(* CODESYS project mobject-graph-plc-pack.library
   Company: mobject
   DefaultNamespace: mobject-graph-plc-pack
   Version: 0.17.0
   Placeholder: mobject-graph-plc-pack
   Author: mobject dev team
   Title: mobject-graph-plc-pack

Project tree, tasks and I/O mapping:
  libraries: mobject-core, 0.7.0 (mobject); mobject-graph, 0.16.0 (mobject); Tc2_Standard, * (Beckhoff Automation GmbH); Tc2_System, * (Beckhoff Automation GmbH); Tc2_Utilities, * (Beckhoff Automation GmbH); Tc3_Module, * (Beckhoff Automation GmbH)
  Datatypes/
    Alias/
      function block _FLOAT [ST]: SetBaseDatatypeReference, Address, ClearReference, Size, FB_init, Clone, Identifier, MakeReferenceTo, TryMakeReferenceTo, Value
      function block _HRESULT [ST]: SetBaseDatatypeReference, Address, ClearReference, Size, FB_init, Clone, Identifier, MakeReferenceTo, TryMakeReferenceTo, Value
    Arrays/
      function block _Array0To7OfByte [ST]: FB_init, OnSerializeArrayValues, SetElementReference, TryDeserializeArrayValues, Address, BaseDatatype, ClearReference, Size, TryGetElementAsDatatypeByIndex, TryGetLowerBound, TryGetUpperBound, Clone, MakeReferenceTo, TryMakeReferenceTo, Value
    Enums/
      function block _E_TcEventClass [ST]: SetBaseDatatypeReference, Address, ClearReference, Size, FB_init, AddLocalEnumeration, IsEnumeratorValueEqual, Clone, Identifier, MakeReferenceTo, TryMakeReferenceTo, Value
    Structs/
      function block _GUID [ST]: Address, ClearReference, Size, FB_init, SetMemberReference, Clone, Identifier, IsValidGuidString, MakeReferenceTo, TryDeserializeFrom, TryMakeReferenceTo, Value, Data1, Data2, Data3, Data4, ToString, TryFromString
      function block _TIMESTRUCT [ST]: Address, ClearReference, Size, FB_init, SetMemberReference, Clone, Identifier, MakeReferenceTo, TryMakeReferenceTo, Value, wDay, wDayOfWeek, wHour, wMilliseconds, wMinute, wMonth, wSecond, wYear
    function block PlcDatatypePack [ST]: RegisterWithDatatypes
  Nodes/
    Converter/
      BOOL_TO_/
      BYTE_TO_/
      DATE_TO_/
      DINT_TO_/
        function block Node_DINT_TO_LREAL [ST]: FB_init, Clone, OnExecute
        function block Node_DINT_TO_REAL [ST]: FB_init, Clone, OnExecute
      DT_TO_/
      DWORD_TO_/
      INT_TO_/
      LINT_TO_/
      LREAL_TO_/
        function block Node_LREAL_TO_DINT [ST]: FB_init, Clone, OnExecute
        function block Node_LREAL_TO_UDINT [ST]: FB_init, Clone, OnExecute
      LWORD_TO_/
      REAL_TO_/
        function block Node_REAL_TO_DINT [ST]: FB_init, Clone, OnExecute
        function block Node_REAL_TO_UDINT [ST]: FB_init, Clone, OnExecute
      SINT_TO_/
      STRING_TO_/
      TIME_TO_/
      TOD_TO_/
      UDINT_TO_/
        function block Node_UDINT_TO_LREAL [ST]: FB_init, Clone, OnExecute
        function block Node_UDINT_TO_REAL [ST]: FB_init, Clone, OnExecute
      UINT_TO_/
      ULINT_TO_/
      USINT_TO_/
      WORD_TO_/
    Hardware/
      Digital/
        function block Node_DigitalInput [ST]: FB_init, OnExecute
        function block Node_DigitalOutput [ST]: FB_init, OnExecute
    Logic/
      function block Node_AND [ST]: FB_init, Clone, OnExecute
      function block Node_NAND [ST]: FB_init, Clone, OnExecute
      function block Node_NOR [ST]: FB_init, Clone, OnExecute
      function block Node_NOT [ST]: FB_init, Clone, OnExecute
      function block Node_OR [ST]: FB_init, Clone, OnExecute
      function block Node_XNOR [ST]: FB_init, Clone, OnExecute
      function block Node_XOR [ST]: FB_init, Clone, OnExecute
    TwinCAT/
      function block Node_TwinCATStatus [ST]: FB_init, Clone, OnExecute
    function block PlcNodePack [ST]: RegisterWithNodeFactory
  function block PlcPack [ST]: Register
*)

// Datatypes/Alias/_FLOAT
{attribute 'linkalways'} 
{attribute 'no_explicit_call' := 'This FB is a CLASS and must be accessed using methods or properties'}
{attribute 'enable_dynamic_creation'}
FUNCTION_BLOCK _FLOAT EXTENDS AliasDatatypeBase
VAR
	localData : FLOAT;
	activeData : REFERENCE TO FLOAT REF= localData;
	aliasBaseDatatype : _LREAL(localData);
END_VAR

METHOD PROTECTED SetBaseDatatypeReference
VAR_INPUT
END_VAR
aliasBaseDatatype.MakeReferenceTo(activeData);
END_METHOD

PROPERTY PUBLIC Address : PVOID
GET
Address := ADR(activeData);
END_GET
END_PROPERTY

METHOD PUBLIC ClearReference
VAR_INPUT
END_VAR
activeData REF= localData;
SetBaseDatatypeReference();
END_METHOD

PROPERTY PUBLIC Size : UDINT
GET
Size := SIZEOF(activeData);
END_GET
END_PROPERTY

METHOD FB_init : BOOL
VAR_INPUT
	bInitRetains : BOOL; // if TRUE, the retain variables are initialized (warm start / cold start)
	bInCopyCode : BOOL;  // if TRUE, the instance afterwards gets moved into the copy code (online change)
	InitialValue : FLOAT;
END_VAR
localData := InitialValue;
SetBaseDatatypeReference();
AddBaseDatatype(aliasBaseDatatype);
END_METHOD

METHOD PUBLIC Clone : I_Datatype
VAR
    pClone : POINTER TO _FLOAT;
END_VAR
pClone := __NEW(_FLOAT(InitialValue := Value));
Clone := pClone^;
END_METHOD

PROPERTY PUBLIC Identifier : T_MAXSTRING
GET
Identifier := 'FLOAT';
END_GET
END_PROPERTY

METHOD PUBLIC MakeReferenceTo
VAR_INPUT
	ReferenceTarget : REFERENCE TO FLOAT;
END_VAR
activeData REF= ReferenceTarget;
SetBaseDatatypeReference();
END_METHOD

METHOD TryMakeReferenceTo : BOOL
VAR_INPUT
	Target : I_Datatype;
END_VAR
VAR
	pTargetData : POINTER TO FLOAT;
END_VAR
IF NOT IsEquivalentTo(Target) THEN
	RETURN;
END_IF

pTargetData := Target.Address;
activeData REF= pTargetData^;
SetBaseDatatypeReference();
TryMakeReferenceTo := TRUE;
END_METHOD

PROPERTY PUBLIC Value : REFERENCE TO FLOAT
GET
Value REF= activeData;
END_GET
END_PROPERTY

END_FUNCTION_BLOCK

// Datatypes/Alias/_HRESULT
{attribute 'linkalways'} 
{attribute 'no_explicit_call' := 'This FB is a CLASS and must be accessed using methods or properties'}
{attribute 'enable_dynamic_creation'}
FUNCTION_BLOCK _HRESULT EXTENDS AliasDatatypeBase
VAR
	localData : HRESULT;
	activeData : REFERENCE TO HRESULT REF= localData;
	aliasBaseDatatype : _DINT(localData);
END_VAR

METHOD PROTECTED SetBaseDatatypeReference
VAR_INPUT
END_VAR
aliasBaseDatatype.MakeReferenceTo(activeData);
END_METHOD

PROPERTY PUBLIC Address : PVOID
GET
Address := ADR(activeData);
END_GET
END_PROPERTY

METHOD PUBLIC ClearReference
VAR_INPUT
END_VAR
activeData REF= localData;
SetBaseDatatypeReference();
END_METHOD

PROPERTY PUBLIC Size : UDINT
GET
Size := SIZEOF(activeData);
END_GET
END_PROPERTY

METHOD FB_init : BOOL
VAR_INPUT
	bInitRetains : BOOL; // if TRUE, the retain variables are initialized (warm start / cold start)
	bInCopyCode : BOOL;  // if TRUE, the instance afterwards gets moved into the copy code (online change)
	InitialValue : HRESULT;
END_VAR
localData := InitialValue;
SetBaseDatatypeReference();
AddBaseDatatype(aliasBaseDatatype);
END_METHOD

METHOD PUBLIC Clone : I_Datatype
VAR
    pClone : POINTER TO _HRESULT;
END_VAR
pClone := __NEW(_HRESULT(InitialValue := Value));
Clone := pClone^;
END_METHOD

PROPERTY PUBLIC Identifier : T_MAXSTRING
GET
Identifier := 'HRESULT';
END_GET
END_PROPERTY

METHOD PUBLIC MakeReferenceTo
VAR_INPUT
	ReferenceTarget : REFERENCE TO HRESULT;
END_VAR
activeData REF= ReferenceTarget;
SetBaseDatatypeReference();
END_METHOD

METHOD TryMakeReferenceTo : BOOL
VAR_INPUT
	Target : I_Datatype;
END_VAR
VAR
	pTargetData : POINTER TO HRESULT;
END_VAR
IF NOT IsEquivalentTo(Target) THEN
	RETURN;
END_IF

pTargetData := Target.Address;
activeData REF= pTargetData^;
SetBaseDatatypeReference();
TryMakeReferenceTo := TRUE;
END_METHOD

PROPERTY PUBLIC Value : REFERENCE TO HRESULT
GET
Value REF= activeData;
END_GET
END_PROPERTY

END_FUNCTION_BLOCK

// Datatypes/Arrays/_Array0To7OfByte
{attribute 'linkalways'} 
{attribute 'no_explicit_call' := 'This FB is a CLASS and must be accessed using methods or properties'}
{attribute 'enable_dynamic_creation'}
FUNCTION_BLOCK _Array0To7OfByte EXTENDS ArrayDatatypeBase_1D
VAR CONSTANT
	lBound : DINT := 0;
	uBound : DINT := 7;
END_VAR
VAR
	localData : ARRAY [lBound..uBound] OF BYTE;
	activeData : REFERENCE TO ARRAY [lBound..uBound] OF BYTE REF= localData;
	elements : ARRAY [lBound..uBound] OF _BYTE(0);
	baseType : _BYTE(0);
END_VAR

METHOD FB_init : BOOL
VAR_INPUT
	bInitRetains : BOOL; // if TRUE, the retain variables are initialized (warm start / cold start)
	bInCopyCode : BOOL;  // if TRUE, the instance afterwards gets moved into the copy code (online change)
END_VAR
SetElementReference();
END_METHOD

METHOD PROTECTED OnSerializeArrayValues
VAR_INPUT
	Serializer : I_Serializer;
END_VAR
VAR
	i : DINT;
END_VAR
FOR i := lBound TO uBound DO
	elements[i].SerializeWith(Serializer);
END_FOR
END_METHOD

METHOD PROTECTED SetElementReference
VAR_INPUT
END_VAR
VAR
	i : DINT;
END_VAR
FOR i := lBound TO uBound DO
	elements[i].MakeReferenceTo(activeData[i]);
END_FOR
END_METHOD

METHOD PROTECTED TryDeserializeArrayValues : BOOL
VAR_INPUT
	Deserializer : I_Deserializer;
	Feedback : I_DeserializerFeedback;
END_VAR
VAR
	enumerator : I_DeserializerArrayForwardEnumerator;
	i : DINT;
END_VAR
enumerator := Deserializer.GetArrayEnumerator();
i := lBound;

WHILE enumerator.MoveNext() AND i <= uBound DO
	
	IF NOT elements[i].TryDeserializeFrom(enumerator.Current, Feedback) THEN
		EXIT;
	END_IF
	i := i + 1;

END_WHILE
enumerator.Dispose();
END_METHOD

PROPERTY PUBLIC Address : PVOID
GET
Address := ADR(activeData);
END_GET
END_PROPERTY

PROPERTY PUBLIC BaseDatatype : I_Datatype
GET
BaseDatatype := baseType;
END_GET
END_PROPERTY

METHOD PUBLIC ClearReference
VAR_INPUT
END_VAR
activeData REF= localData;
SetElementReference();
END_METHOD

PROPERTY PUBLIC Size : UDINT
GET
Size := SIZEOF(activeData);
END_GET
END_PROPERTY

METHOD PUBLIC TryGetElementAsDatatypeByIndex : BOOL
VAR_INPUT
	Index : DINT;
	Destination : REFERENCE TO I_Datatype;
END_VAR
IF Index < lbound OR Index > ubound THEN
	RETURN;
END_IF

Destination := elements[Index];
TryGetElementAsDatatypeByIndex := TRUE;
END_METHOD

METHOD PUBLIC TryGetLowerBound : BOOL
VAR_INPUT
	Dimention : UDINT;
	Destination : REFERENCE TO DINT;
END_VAR
IF Dimention = 1 THEN
	Destination := lBound;
	TryGetLowerBound := TRUE;
END_IF
END_METHOD

METHOD PUBLIC TryGetUpperBound : BOOL
VAR_INPUT
	Dimention : UDINT;
	Destination : REFERENCE TO DINT;
END_VAR
IF Dimention = 1 THEN
	Destination := uBound;
	TryGetUpperBound := TRUE;
END_IF
END_METHOD

METHOD PUBLIC Clone : I_Datatype
VAR
    pClone : POINTER TO _Array0To7OfByte;
END_VAR
pClone := __NEW(_Array0To7OfByte());
pClone^.Value := Value;
Clone := pClone^;
END_METHOD

METHOD PUBLIC MakeReferenceTo
VAR_INPUT
	ReferenceTarget : REFERENCE TO ARRAY [lBound..uBound] OF BYTE;
END_VAR
activeData REF= ReferenceTarget;
SetElementReference();
END_METHOD

METHOD TryMakeReferenceTo : BOOL
VAR_INPUT
	Target : I_Datatype;
END_VAR
VAR
	pTargetData : POINTER TO ARRAY [lBound..uBound] OF BYTE;
END_VAR
IF NOT IsEquivalentTo(Target) THEN
	RETURN;
END_IF

pTargetData := Target.Address;
activeData REF= pTargetData^;
SetElementReference();
TryMakeReferenceTo := TRUE;
END_METHOD

PROPERTY PUBLIC Value : REFERENCE TO ARRAY [lBound..uBound] OF BYTE;
GET
Value ref= activeData;
END_GET
END_PROPERTY

END_FUNCTION_BLOCK

// Datatypes/Enums/_E_TcEventClass
{attribute 'linkalways'} 
{attribute 'no_explicit_call' := 'This FB is a CLASS and must be accessed using methods or properties'}
{attribute 'enable_dynamic_creation'}
FUNCTION_BLOCK _E_TcEventClass EXTENDS EnumDatatypeBase
VAR
	localData : E_TcEventClass;
	activeData : REFERENCE TO E_TcEventClass;
	enumBaseDatatype : _UINT(localData);
END_VAR

METHOD PROTECTED SetBaseDatatypeReference
VAR_INPUT
END_VAR
enumBaseDatatype.MakeReferenceTo(activeData);
END_METHOD

PROPERTY PUBLIC Address : PVOID
GET
Address := ADR(activeData);
END_GET
END_PROPERTY

METHOD PUBLIC ClearReference
VAR_INPUT
END_VAR
activeData REF= localData;
SetBaseDatatypeReference();
END_METHOD

PROPERTY PUBLIC Size : UDINT
GET
Size := SIZEOF(activeData);
END_GET
END_PROPERTY

METHOD FB_init : BOOL
VAR_INPUT
	bInitRetains : BOOL; // if TRUE, the retain variables are initialized (warm start / cold start)
	bInCopyCode : BOOL;  // if TRUE, the instance afterwards gets moved into the copy code (online change)
	InitialValue : E_TcEventClass;
END_VAR
localData := InitialValue;
AddBaseDatatype(enumBaseDatatype);
ClearReference();

AddLocalEnumeration('TCEVENTCLASS_NONE', E_TcEventClass.TCEVENTCLASS_NONE);
AddLocalEnumeration('TCEVENTCLASS_MAINTENANCE', E_TcEventClass.TCEVENTCLASS_MAINTENANCE);
AddLocalEnumeration('TCEVENTCLASS_MESSAGE', E_TcEventClass.TCEVENTCLASS_MESSAGE);
AddLocalEnumeration('TCEVENTCLASS_HINT', E_TcEventClass.TCEVENTCLASS_HINT);
AddLocalEnumeration('TCEVENTCLASS_STATEINFO', E_TcEventClass.TCEVENTCLASS_STATEINFO);
AddLocalEnumeration('TCEVENTCLASS_INSTRUCTION', E_TcEventClass.TCEVENTCLASS_INSTRUCTION);
AddLocalEnumeration('TCEVENTCLASS_WARNING', E_TcEventClass.TCEVENTCLASS_WARNING);
AddLocalEnumeration('TCEVENTCLASS_ALARM', E_TcEventClass.TCEVENTCLASS_ALARM);
AddLocalEnumeration('TCEVENTCLASS_PARAMERROR', E_TcEventClass.TCEVENTCLASS_PARAMERROR);
END_METHOD

METHOD PRIVATE AddLocalEnumeration
VAR_INPUT
	Enumeration : T_MAXSTRING;
	Value : E_TcEventClass;
END_VAR
AddEnumeration(Enumeration, Value);
END_METHOD

METHOD IsEnumeratorValueEqual : BOOL
VAR_INPUT
	Enumerator : I_KeyValueForwardEnumerator;
END_VAR
VAR
	storedValue : E_TcEventClass;
END_VAR
IF NOT Enumerator.TryGet(storedValue) THEN
	RETURN;
END_IF

IsEnumeratorValueEqual := storedValue = activeData;
END_METHOD

METHOD PUBLIC Clone : I_Datatype
VAR
    pClone : POINTER TO _E_TcEventClass;
END_VAR
pClone := __NEW(_E_TcEventClass(InitialValue := Value));
Clone := pClone^;
END_METHOD

PROPERTY PUBLIC Identifier : T_MAXSTRING
GET
Identifier := 'E_TcEventClass';
END_GET
END_PROPERTY

METHOD PUBLIC MakeReferenceTo
VAR_INPUT
	ReferenceTarget : REFERENCE TO E_TcEventClass;
END_VAR
activeData REF= ReferenceTarget;
SetBaseDatatypeReference();
END_METHOD

METHOD TryMakeReferenceTo : BOOL
VAR_INPUT
	Target : I_Datatype;
END_VAR
VAR
	pTargetData : POINTER TO E_TcEventClass;
END_VAR
IF NOT IsEquivalentTo(Target) THEN
	RETURN;
END_IF

pTargetData := Target.Address;
activeData REF= pTargetData^;
SetBaseDatatypeReference();
TryMakeReferenceTo := TRUE;
END_METHOD

PROPERTY PUBLIC Value : REFERENCE TO E_TcEventClass
GET
Value REF= activeData;
END_GET
END_PROPERTY

END_FUNCTION_BLOCK

// Datatypes/Structs/_GUID
{attribute 'linkalways'} 
{attribute 'no_explicit_call' := 'This FB is a CLASS and must be accessed using methods or properties'}
{attribute 'enable_dynamic_creation'}
FUNCTION_BLOCK _GUID EXTENDS StructuredDatatypeBase
VAR
	localData : GUID;
	activeData : REFERENCE TO GUID REF= localData;
	_data1 : _DWORD(localData.data1);
	_data2 : _WORD(localData.data2);
    _data3 : _WORD(localData.data3);
	_data4 : _Array0To7OfByte();
END_VAR

PROPERTY PUBLIC Address : PVOID
GET
Address := ADR(activeData);
END_GET
END_PROPERTY

METHOD PUBLIC ClearReference
VAR_INPUT
END_VAR
activeData REF= localData;
SetMemberReference();
END_METHOD

PROPERTY PUBLIC Size : UDINT
GET
Size := SIZEOF(activeData);
END_GET
END_PROPERTY

METHOD FB_init : BOOL
VAR_INPUT
	bInitRetains : BOOL; // if TRUE, the retain variables are initialized (warm start / cold start)
	bInCopyCode : BOOL;  // if TRUE, the instance afterwards gets moved into the copy code (online change)
END_VAR
SetMemberReference();
AddMember('Data1',_data1);
AddMember('Data2',_data2);
AddMember('Data3',_data3);
AddMember('Data4',_data4);
END_METHOD

METHOD PROTECTED SetMemberReference
VAR_INPUT
END_VAR
_data1.MakeReferenceTo(activeData.Data1);
_data2.MakeReferenceTo(activeData.Data2);
_data3.MakeReferenceTo(activeData.Data3);
_data4.MakeReferenceTo(activeData.Data4);
END_METHOD

METHOD PUBLIC Clone : I_Datatype
VAR
    pClone : POINTER TO _GUID;
END_VAR
pClone := __NEW(_GUID());
pClone^.Value := Value;
Clone := pClone^;
END_METHOD

PROPERTY PUBLIC Identifier : T_MAXSTRING
GET
Identifier := 'GUID';
END_GET
END_PROPERTY

METHOD PROTECTED IsValidGuidString : BOOL
VAR_INPUT
	GuidAsString : STRING;
END_VAR
VAR
	position : INT;
	stringIndex : INT;
	dashCount : INT := 0;
END_VAR
VAR CONSTANT
	CHARACTER_HYPHEN : BYTE := 16#2D;
	CHARACTER_0 : BYTE := 16#30;
	CHARACTER_9 : BYTE := 16#39;
	CHARACTER_A : BYTE := 16#41;
	CHARACTER_F : BYTE := 16#46;
	CHARACTER_LCASE_A : BYTE := 16#61;
	CHARACTER_LCASE_F : BYTE := 16#66;
END_VAR
// Check the overall length of the string (36 including 4 dashes)
IF LEN(GuidAsString) <> 36 THEN
	RETURN;
END_IF

// Check each character
FOR position := 1 TO 36 DO
	stringIndex := position - 1; 
	CASE position OF
		9, 14, 19, 24:
			// Dashes should be at positions 9, 14, 19, 24
			IF GuidAsString[stringIndex] <> CHARACTER_HYPHEN THEN
				RETURN;
			ELSE
				dashCount := dashCount + 1;
			END_IF
		ELSE
			// All other positions should contain hex digits (0-9, A-F, a-f)
			IF NOT ((GuidAsString[stringIndex] >= CHARACTER_0 AND GuidAsString[stringIndex] <= CHARACTER_9) OR 
				(GuidAsString[stringIndex] >= CHARACTER_A AND GuidAsString[stringIndex] <= CHARACTER_F) OR 
				(GuidAsString[stringIndex] >= CHARACTER_LCASE_A AND GuidAsString[stringIndex] <= CHARACTER_LCASE_F)) THEN
				RETURN;
			END_IF
	END_CASE
END_FOR

// Ensure exactly four dashes are present
IF dashCount = 4 THEN
	IsValidGuidString := TRUE;
END_IF
END_METHOD

METHOD PUBLIC MakeReferenceTo
VAR_INPUT
	ReferenceTarget : REFERENCE TO GUID;
END_VAR
activeData REF= ReferenceTarget;
SetMemberReference();
END_METHOD

METHOD TryDeserializeFrom : BOOL
VAR_INPUT
	Deserializer : I_Deserializer;
	Feedback : I_DeserializerFeedback;
END_VAR
VAR
	localFeedback : DeserializerFeedback;
	guidAsString : T_MAXSTRING;
END_VAR
// this customized version of TryDeserializeFrom allows for the use of string guids. 
// if a string is not found, then it will try to deserialize from an object.
IF Deserializer.TryGetString(guidAsString, localFeedback) THEN	
	IF TryFromString(guidAsString) THEN
		TryDeserializeFrom := TRUE;
		RETURN;
	END_IF
	
	Feedback.LogDeserializationFailedError('Invalid GUID String');	
	RETURN;
END_IF

TryDeserializeFrom := SUPER^.TryDeserializeFrom(Deserializer, Feedback);
END_METHOD

METHOD TryMakeReferenceTo : BOOL
VAR_INPUT
	Target : I_Datatype;
END_VAR
VAR
	pTargetData : POINTER TO GUID;
END_VAR
IF NOT IsEquivalentTo(Target) THEN
	RETURN;
END_IF

pTargetData := Target.Address;
activeData REF= pTargetData^;
SetMemberReference();
TryMakeReferenceTo := TRUE;
END_METHOD

PROPERTY PUBLIC Value : REFERENCE TO GUID
GET
Value REF= activeData;
END_GET
END_PROPERTY

PROPERTY PUBLIC Data1 : REFERENCE TO _DWORD
GET
Data1 REF= _data1;
END_GET
END_PROPERTY

PROPERTY PUBLIC Data2 : REFERENCE TO _WORD
GET
Data2 REF= _data2;
END_GET
END_PROPERTY

PROPERTY PUBLIC Data3 : REFERENCE TO _WORD
GET
Data3 REF= _data3;
END_GET
END_PROPERTY

PROPERTY PUBLIC Data4 : REFERENCE TO _Array0To7OfByte
GET
Data4 REF= _data4;
END_GET
END_PROPERTY

METHOD PUBLIC ToString : T_MAXSTRING
VAR_INPUT
END_VAR
ToString := GUID_TO_STRING(activeData);
END_METHOD

METHOD PUBLIC TryFromString : BOOL;
VAR_INPUT
	GuidAsString : T_MAXSTRING;
END_VAR
IF NOT IsValidGuidString(GuidAsString) THEN
	RETURN;
END_IF

activeData := STRING_TO_GUID(GuidAsString);
TryFromString := true;
END_METHOD

END_FUNCTION_BLOCK

// Datatypes/Structs/_TIMESTRUCT
{attribute 'linkalways'} 
{attribute 'no_explicit_call' := 'This FB is a CLASS and must be accessed using methods or properties'}
{attribute 'enable_dynamic_creation'}
FUNCTION_BLOCK _TIMESTRUCT EXTENDS StructuredDatatypeBase
VAR
	localData : TIMESTRUCT;
	activeData : REFERENCE TO TIMESTRUCT REF= localData;
	_wYear : _WORD(localData.wYear);
	_wMonth : _WORD(localData.wMonth);
	_wDayOfWeek : _WORD(localData.wDayOfWeek);
	_wDay : _WORD(localData.wDay);
	_wHour : _WORD(localData.wHour);
	_wMinute : _WORD(localData.wMinute);
	_wSecond : _WORD(localData.wSecond);
	_wMilliseconds : _WORD(localData.wMilliseconds);
END_VAR

PROPERTY PUBLIC Address : PVOID
GET
Address := ADR(activeData);
END_GET
END_PROPERTY

METHOD PUBLIC ClearReference
VAR_INPUT
END_VAR
activeData REF= localData;
SetMemberReference();
END_METHOD

PROPERTY PUBLIC Size : UDINT
GET
Size := SIZEOF(activeData);
END_GET
END_PROPERTY

METHOD FB_init : BOOL
VAR_INPUT
	bInitRetains : BOOL; // if TRUE, the retain variables are initialized (warm start / cold start)
	bInCopyCode : BOOL;  // if TRUE, the instance afterwards gets moved into the copy code (online change)
END_VAR
SetMemberReference();
AddMember('wYear',_wYear);
AddMember('wMonth',_wMonth);
AddMember('wDayOfWeek',_wDayOfWeek);
AddMember('wDay',_wDay);
AddMember('wHour',_wHour);
AddMember('wMinute',_wMinute);
AddMember('wSecond',_wSecond);
AddMember('wMilliseconds',_wMilliseconds);
END_METHOD

METHOD PROTECTED SetMemberReference
VAR_INPUT
END_VAR
_wYear.MakeReferenceTo(activeData.wYear);
_wMonth.MakeReferenceTo(activeData.wMonth);
_wDayOfWeek.MakeReferenceTo(activeData.wDayOfWeek);
_wDay.MakeReferenceTo(activeData.wDay);
_wHour.MakeReferenceTo(activeData.wHour);
_wMinute.MakeReferenceTo(activeData.wMinute);
_wSecond.MakeReferenceTo(activeData.wSecond);
_wMilliseconds.MakeReferenceTo(activeData.wMilliseconds);
END_METHOD

METHOD PUBLIC Clone : I_Datatype
VAR
    pClone : POINTER TO _TIMESTRUCT;
END_VAR
pClone := __NEW(_TIMESTRUCT());
pClone^.Value := Value;
Clone := pClone^;
END_METHOD

PROPERTY PUBLIC Identifier : T_MAXSTRING
GET
Identifier := 'TIMESTRUCT';
END_GET
END_PROPERTY

METHOD PUBLIC MakeReferenceTo
VAR_INPUT
	ReferenceTarget : REFERENCE TO TIMESTRUCT;
END_VAR
activeData REF= ReferenceTarget;
SetMemberReference();
END_METHOD

METHOD TryMakeReferenceTo : BOOL
VAR_INPUT
	Target : I_Datatype;
END_VAR
VAR
	pTargetData : POINTER TO TIMESTRUCT;
END_VAR
IF NOT IsEquivalentTo(Target) THEN
	RETURN;
END_IF

pTargetData := Target.Address;
activeData REF= pTargetData^;
SetMemberReference();
TryMakeReferenceTo := TRUE;
END_METHOD

PROPERTY PUBLIC Value : REFERENCE TO TIMESTRUCT
GET
Value REF= activeData;
END_GET
END_PROPERTY

PROPERTY PUBLIC wDay : Reference to _WORD
GET
wDay REF= _wDay;
END_GET
END_PROPERTY

PROPERTY PUBLIC wDayOfWeek : Reference to _WORD
GET
wDayOfWeek REF= _wDayOfWeek;
END_GET
END_PROPERTY

PROPERTY PUBLIC wHour : Reference to _WORD
GET
wHour REF= _wHour;
END_GET
END_PROPERTY

PROPERTY PUBLIC wMilliseconds : Reference to _WORD
GET
wMilliseconds REF= _wMilliseconds;
END_GET
END_PROPERTY

PROPERTY PUBLIC wMinute : Reference to _WORD
GET
wMinute REF= _wMinute;
END_GET
END_PROPERTY

PROPERTY PUBLIC wMonth : Reference to _WORD
GET
wMonth REF= _wMonth;
END_GET
END_PROPERTY

PROPERTY PUBLIC wSecond : Reference to _WORD
GET
wSecond REF= _wSecond;
END_GET
END_PROPERTY

PROPERTY PUBLIC wYear : Reference to _WORD
GET
wYear REF= _wYear;
END_GET
END_PROPERTY

END_FUNCTION_BLOCK

// Datatypes/PlcDatatypePack
{attribute 'linkalways'} 
{attribute 'no_explicit_call' := 'This FB is a CLASS and must be accessed using methods or properties'}
{attribute 'enable_dynamic_creation'}
FUNCTION_BLOCK PlcDatatypePack
VAR
	
	// alias
    _float : _FLOAT(0.0);
	_hresult : _HRESULT(0);

	// enums
	_e_TcEventClass : _E_TcEventClass(E_TcEventClass.TCEVENTCLASS_NONE);
	
	// structures
	_timestruct : _TIMESTRUCT();
	
END_VAR

METHOD RegisterWithDatatypes
VAR_INPUT
	Datatypes : I_Datatypes;
END_VAR
// alias
Datatypes.RegisterDatatype(_float);
Datatypes.RegisterDatatype(_hresult);

// enums
Datatypes.RegisterDatatype(_e_TcEventClass);

// structures
Datatypes.RegisterDatatype(_timestruct);
END_METHOD

END_FUNCTION_BLOCK

// Nodes/Converter/DINT_TO_/Node_DINT_TO_LREAL
{attribute 'linkalways'} 
{attribute 'no_explicit_call' := 'This FB is a CLASS and must be accessed using methods or properties'}
{attribute 'enable_dynamic_creation'}
FUNCTION_BLOCK FINAL Node_DINT_TO_LREAL EXTENDS Node
VAR
	in : _DINT(0);
	out : _LREAL(0.0);
	success : _BOOL(FALSE);
END_VAR

METHOD FB_init : BOOL
VAR_INPUT
	bInitRetains : BOOL; // if TRUE, the retain variables are initialized (warm start / cold start)
	bInCopyCode : BOOL;  // if TRUE, the instance afterwards gets moved into the copy code (online change)
END_VAR
AddParameter('in', in);
AddOutput('out', out);
AddOutput('success', success);
END_METHOD

METHOD PUBLIC  Clone : I_Node
VAR
	pNode : POINTER TO Node_DINT_TO_LREAL;
END_VAR
pNode := __NEW(Node_DINT_TO_LREAL);
Clone := pNode^;
END_METHOD

METHOD PROTECTED OnExecute
VAR
END_VAR
success.Value := TryConvert_DINT_TO_LREAL(in.Value, out.Value);
END_METHOD

END_FUNCTION_BLOCK

// Nodes/Converter/DINT_TO_/Node_DINT_TO_REAL
{attribute 'linkalways'} 
{attribute 'no_explicit_call' := 'This FB is a CLASS and must be accessed using methods or properties'}
{attribute 'enable_dynamic_creation'}
FUNCTION_BLOCK FINAL Node_DINT_TO_REAL EXTENDS Node
VAR
	in : _DINT(0);
	out : _REAL(0.0);
	success : _BOOL(FALSE);
END_VAR

METHOD FB_init : BOOL
VAR_INPUT
	bInitRetains : BOOL; // if TRUE, the retain variables are initialized (warm start / cold start)
	bInCopyCode : BOOL;  // if TRUE, the instance afterwards gets moved into the copy code (online change)
END_VAR
AddParameter('in', in);
AddOutput('out', out);
AddOutput('success', success);
END_METHOD

METHOD PUBLIC  Clone : I_Node
VAR
	pNode : POINTER TO Node_DINT_TO_REAL;
END_VAR
pNode := __NEW(Node_DINT_TO_REAL);
Clone := pNode^;
END_METHOD

METHOD PROTECTED OnExecute
VAR
END_VAR
success.Value := TryConvert_DINT_TO_REAL(in.Value, out.Value);
END_METHOD

END_FUNCTION_BLOCK

// Nodes/Converter/LREAL_TO_/Node_LREAL_TO_DINT
{attribute 'linkalways'} 
{attribute 'no_explicit_call' := 'This FB is a CLASS and must be accessed using methods or properties'}
{attribute 'enable_dynamic_creation'}
FUNCTION_BLOCK FINAL Node_LREAL_TO_DINT EXTENDS Node
VAR
	in : _LREAL(0.0);
	out : _DINT(0);
	success : _BOOL(FALSE);
END_VAR

METHOD FB_init : BOOL
VAR_INPUT
	bInitRetains : BOOL; // if TRUE, the retain variables are initialized (warm start / cold start)
	bInCopyCode : BOOL;  // if TRUE, the instance afterwards gets moved into the copy code (online change)
END_VAR
AddParameter('in', in);
AddOutput('out', out);
AddOutput('success', success);
END_METHOD

METHOD PUBLIC  Clone : I_Node
VAR
	pNode : POINTER TO Node_LREAL_TO_DINT;
END_VAR
pNode := __NEW(Node_LREAL_TO_DINT);
Clone := pNode^;
END_METHOD

METHOD PROTECTED OnExecute
VAR
END_VAR
success.Value := TryConvert_LREAL_TO_DINT(in.Value, out.Value);
END_METHOD

END_FUNCTION_BLOCK

// Nodes/Converter/LREAL_TO_/Node_LREAL_TO_UDINT
{attribute 'linkalways'} 
{attribute 'no_explicit_call' := 'This FB is a CLASS and must be accessed using methods or properties'}
{attribute 'enable_dynamic_creation'}
FUNCTION_BLOCK FINAL Node_LREAL_TO_UDINT EXTENDS Node
VAR
	in : _LREAL(0.0);
	out : _UDINT(0);
	success : _BOOL(FALSE);
END_VAR

METHOD FB_init : BOOL
VAR_INPUT
	bInitRetains : BOOL; // if TRUE, the retain variables are initialized (warm start / cold start)
	bInCopyCode : BOOL;  // if TRUE, the instance afterwards gets moved into the copy code (online change)
END_VAR
AddParameter('in', in);
AddOutput('out', out);
AddOutput('success', success);
END_METHOD

METHOD PUBLIC  Clone : I_Node
VAR
	pNode : POINTER TO Node_LREAL_TO_UDINT;
END_VAR
pNode := __NEW(Node_LREAL_TO_UDINT);
Clone := pNode^;
END_METHOD

METHOD PROTECTED OnExecute
VAR
END_VAR
success.Value := TryConvert_LREAL_TO_UDINT(in.Value, out.Value);
END_METHOD

END_FUNCTION_BLOCK

// Nodes/Converter/REAL_TO_/Node_REAL_TO_DINT
{attribute 'linkalways'} 
{attribute 'no_explicit_call' := 'This FB is a CLASS and must be accessed using methods or properties'}
{attribute 'enable_dynamic_creation'}
FUNCTION_BLOCK FINAL Node_REAL_TO_DINT EXTENDS Node
VAR
	in : _REAL(0.0);
	out : _DINT(0);
	success : _BOOL(FALSE);
END_VAR

METHOD FB_init : BOOL
VAR_INPUT
	bInitRetains : BOOL; // if TRUE, the retain variables are initialized (warm start / cold start)
	bInCopyCode : BOOL;  // if TRUE, the instance afterwards gets moved into the copy code (online change)
END_VAR
AddParameter('in', in);
AddOutput('out', out);
AddOutput('success', success);
END_METHOD

METHOD PUBLIC  Clone : I_Node
VAR
	pNode : POINTER TO Node_REAL_TO_DINT;
END_VAR
pNode := __NEW(Node_REAL_TO_DINT);
Clone := pNode^;
END_METHOD

METHOD PROTECTED OnExecute
VAR
END_VAR
success.Value := TryConvert_REAL_TO_DINT(in.Value, out.Value);
END_METHOD

END_FUNCTION_BLOCK

// Nodes/Converter/REAL_TO_/Node_REAL_TO_UDINT
{attribute 'linkalways'} 
{attribute 'no_explicit_call' := 'This FB is a CLASS and must be accessed using methods or properties'}
{attribute 'enable_dynamic_creation'}
FUNCTION_BLOCK FINAL Node_REAL_TO_UDINT EXTENDS Node
VAR
	in : _REAL(0.0);
	out : _UDINT(0);
	success : _BOOL(FALSE);
END_VAR

METHOD FB_init : BOOL
VAR_INPUT
	bInitRetains : BOOL; // if TRUE, the retain variables are initialized (warm start / cold start)
	bInCopyCode : BOOL;  // if TRUE, the instance afterwards gets moved into the copy code (online change)
END_VAR
AddParameter('in', in);
AddOutput('out', out);
AddOutput('success', success);
END_METHOD

METHOD PUBLIC  Clone : I_Node
VAR
	pNode : POINTER TO Node_REAL_TO_UDINT;
END_VAR
pNode := __NEW(Node_REAL_TO_UDINT);
Clone := pNode^;
END_METHOD

METHOD PROTECTED OnExecute
VAR
END_VAR
success.Value := TryConvert_REAL_TO_UDINT(in.Value, out.Value);
END_METHOD

END_FUNCTION_BLOCK

// Nodes/Converter/UDINT_TO_/Node_UDINT_TO_LREAL
{attribute 'linkalways'} 
{attribute 'no_explicit_call' := 'This FB is a CLASS and must be accessed using methods or properties'}
{attribute 'enable_dynamic_creation'}
FUNCTION_BLOCK FINAL Node_UDINT_TO_LREAL EXTENDS Node
VAR
	in : _UDINT(0);
	out : _LREAL(0.0);
	success : _BOOL(FALSE);
END_VAR

METHOD FB_init : BOOL
VAR_INPUT
	bInitRetains : BOOL; // if TRUE, the retain variables are initialized (warm start / cold start)
	bInCopyCode : BOOL;  // if TRUE, the instance afterwards gets moved into the copy code (online change)
END_VAR
AddParameter('in', in);
AddOutput('out', out);
AddOutput('success', success);
END_METHOD

METHOD PUBLIC  Clone : I_Node
VAR
	pNode : POINTER TO Node_UDINT_TO_LREAL;
END_VAR
pNode := __NEW(Node_UDINT_TO_LREAL);
Clone := pNode^;
END_METHOD

METHOD PROTECTED OnExecute
VAR
END_VAR
success.Value := TryConvert_UDINT_TO_LREAL(in.Value, out.Value);
END_METHOD

END_FUNCTION_BLOCK

// Nodes/Converter/UDINT_TO_/Node_UDINT_TO_REAL
{attribute 'linkalways'} 
{attribute 'no_explicit_call' := 'This FB is a CLASS and must be accessed using methods or properties'}
{attribute 'enable_dynamic_creation'}
FUNCTION_BLOCK FINAL Node_UDINT_TO_REAL EXTENDS Node
VAR
	in : _UDINT(0);
	out : _REAL(0.0);
	success : _BOOL(FALSE);
END_VAR

METHOD FB_init : BOOL
VAR_INPUT
	bInitRetains : BOOL; // if TRUE, the retain variables are initialized (warm start / cold start)
	bInCopyCode : BOOL;  // if TRUE, the instance afterwards gets moved into the copy code (online change)
END_VAR
AddParameter('in', in);
AddOutput('out', out);
AddOutput('success', success);
END_METHOD

METHOD PUBLIC  Clone : I_Node
VAR
	pNode : POINTER TO Node_UDINT_TO_REAL;
END_VAR
pNode := __NEW(Node_UDINT_TO_REAL);
Clone := pNode^;
END_METHOD

METHOD PROTECTED OnExecute
VAR
END_VAR
success.Value := TryConvert_UDINT_TO_REAL(in.Value, out.Value);
END_METHOD

END_FUNCTION_BLOCK

// Nodes/Hardware/Digital/Node_DigitalInput
{attribute 'linkalways'} 
{attribute 'no_explicit_call' := 'This FB is a CLASS and must be accessed using methods or properties'}
{attribute 'enable_dynamic_creation'}
FUNCTION_BLOCK FINAL Node_DigitalInput EXTENDS HardwareNode
VAR
	input AT %I* : BOOL;
	out : _BOOL(FALSE);
END_VAR

METHOD FB_init : BOOL
VAR_INPUT
	bInitRetains : BOOL; // if TRUE, the retain variables are initialized (warm start / cold start)
	bInCopyCode : BOOL;  // if TRUE, the instance afterwards gets moved into the copy code (online change)
END_VAR
AddOutput('out', out);
END_METHOD

METHOD PROTECTED OnExecute
VAR
END_VAR
out.Value := input;
END_METHOD

END_FUNCTION_BLOCK

// Nodes/Hardware/Digital/Node_DigitalOutput
{attribute 'linkalways'} 
{attribute 'no_explicit_call' := 'This FB is a CLASS and must be accessed using methods or properties'}
{attribute 'enable_dynamic_creation'}
FUNCTION_BLOCK FINAL Node_DigitalOutput EXTENDS HardwareNode
VAR
	output AT %Q* : BOOL;
	in : _BOOL(FALSE);
END_VAR

METHOD FB_init : BOOL
VAR_INPUT
	bInitRetains : BOOL; // if TRUE, the retain variables are initialized (warm start / cold start)
	bInCopyCode : BOOL;  // if TRUE, the instance afterwards gets moved into the copy code (online change)
END_VAR
AddParameter('in', in);
END_METHOD

METHOD PROTECTED OnExecute
VAR
END_VAR
output := in.Value;
END_METHOD

END_FUNCTION_BLOCK

// Nodes/Logic/Node_AND
{attribute 'linkalways'} 
{attribute 'no_explicit_call' := 'This FB is a CLASS and must be accessed using methods or properties'}
{attribute 'enable_dynamic_creation'}
FUNCTION_BLOCK FINAL Node_AND EXTENDS Node
VAR
	in1 : _BOOL(FALSE);
    in2 : _BOOL(FALSE);
	out : _BOOL(FALSE);
END_VAR

METHOD FB_init : BOOL
VAR_INPUT
	bInitRetains : BOOL; // if TRUE, the retain variables are initialized (warm start / cold start)
	bInCopyCode : BOOL;  // if TRUE, the instance afterwards gets moved into the copy code (online change)
END_VAR
AddParameter('in1', in1);
AddParameter('in2', in2);
AddOutput('out', out);
END_METHOD

METHOD PUBLIC  Clone : I_Node
VAR
	pNode : POINTER TO Node_AND;
END_VAR
pNode := __NEW(Node_AND);
Clone := pNode^;
END_METHOD

METHOD PROTECTED OnExecute
VAR
END_VAR
out.Value := in1.Value AND in2.Value;
END_METHOD

END_FUNCTION_BLOCK

// Nodes/Logic/Node_NAND
{attribute 'linkalways'} 
{attribute 'no_explicit_call' := 'This FB is a CLASS and must be accessed using methods or properties'}
{attribute 'enable_dynamic_creation'}
FUNCTION_BLOCK FINAL Node_NAND EXTENDS Node
VAR
	in1 : _BOOL(FALSE);
    in2 : _BOOL(FALSE);
	out : _BOOL(FALSE);
END_VAR

METHOD FB_init : BOOL
VAR_INPUT
	bInitRetains : BOOL; // if TRUE, the retain variables are initialized (warm start / cold start)
	bInCopyCode : BOOL;  // if TRUE, the instance afterwards gets moved into the copy code (online change)
END_VAR
AddParameter('in1', in1);
AddParameter('in2', in2);
AddOutput('out', out);
END_METHOD

METHOD PUBLIC  Clone : I_Node
VAR
	pNode : POINTER TO Node_NAND;
END_VAR
pNode := __NEW(Node_NAND);
Clone := pNode^;
END_METHOD

METHOD PROTECTED OnExecute
VAR
END_VAR
out.Value := NOT(in1.Value AND in2.Value);
END_METHOD

END_FUNCTION_BLOCK

// Nodes/Logic/Node_NOR
{attribute 'linkalways'} 
{attribute 'no_explicit_call' := 'This FB is a CLASS and must be accessed using methods or properties'}
{attribute 'enable_dynamic_creation'}
FUNCTION_BLOCK FINAL Node_NOR EXTENDS Node
VAR
	in1 : _BOOL(FALSE);
    in2 : _BOOL(FALSE);
	out : _BOOL(FALSE);
END_VAR

METHOD FB_init : BOOL
VAR_INPUT
	bInitRetains : BOOL; // if TRUE, the retain variables are initialized (warm start / cold start)
	bInCopyCode : BOOL;  // if TRUE, the instance afterwards gets moved into the copy code (online change)
END_VAR
AddParameter('in1', in1);
AddParameter('in2', in2);
AddOutput('out', out);
END_METHOD

METHOD PUBLIC  Clone : I_Node
VAR
	pNode : POINTER TO Node_NOR;
END_VAR
pNode := __NEW(Node_NOR);
Clone := pNode^;
END_METHOD

METHOD PROTECTED OnExecute
VAR
END_VAR
out.Value := NOT(in1.Value OR in2.Value);
END_METHOD

END_FUNCTION_BLOCK

// Nodes/Logic/Node_NOT
{attribute 'linkalways'} 
{attribute 'no_explicit_call' := 'This FB is a CLASS and must be accessed using methods or properties'}
{attribute 'enable_dynamic_creation'}
FUNCTION_BLOCK FINAL Node_NOT EXTENDS Node
VAR
	in : _BOOL(FALSE);
	out : _BOOL(FALSE);
END_VAR

METHOD FB_init : BOOL
VAR_INPUT
	bInitRetains : BOOL; // if TRUE, the retain variables are initialized (warm start / cold start)
	bInCopyCode : BOOL;  // if TRUE, the instance afterwards gets moved into the copy code (online change)
END_VAR
AddParameter('in', in);
AddOutput('out', out);
END_METHOD

METHOD PUBLIC  Clone : I_Node
VAR
	pNode : POINTER TO Node_NOT;
END_VAR
pNode := __NEW(Node_NOT);
Clone := pNode^;
END_METHOD

METHOD PROTECTED OnExecute
VAR
END_VAR
out.Value := NOT in.Value;
END_METHOD

END_FUNCTION_BLOCK

// Nodes/Logic/Node_OR
{attribute 'linkalways'} 
{attribute 'no_explicit_call' := 'This FB is a CLASS and must be accessed using methods or properties'}
{attribute 'enable_dynamic_creation'}
FUNCTION_BLOCK FINAL Node_OR EXTENDS Node
VAR
	in1 : _BOOL(FALSE);
    in2 : _BOOL(FALSE);
	out : _BOOL(FALSE);
END_VAR

METHOD FB_init : BOOL
VAR_INPUT
	bInitRetains : BOOL; // if TRUE, the retain variables are initialized (warm start / cold start)
	bInCopyCode : BOOL;  // if TRUE, the instance afterwards gets moved into the copy code (online change)
END_VAR
AddParameter('in1', in1);
AddParameter('in2', in2);
AddOutput('out', out);
END_METHOD

METHOD PUBLIC  Clone : I_Node
VAR
	pNode : POINTER TO Node_OR;
END_VAR
pNode := __NEW(Node_OR);
Clone := pNode^;
END_METHOD

METHOD PROTECTED OnExecute
VAR
END_VAR
out.Value := in1.Value OR in2.Value;
END_METHOD

END_FUNCTION_BLOCK

// Nodes/Logic/Node_XNOR
{attribute 'linkalways'} 
{attribute 'no_explicit_call' := 'This FB is a CLASS and must be accessed using methods or properties'}
{attribute 'enable_dynamic_creation'}
FUNCTION_BLOCK FINAL Node_XNOR EXTENDS Node
VAR
	in1 : _BOOL(FALSE);
    in2 : _BOOL(FALSE);
	out : _BOOL(FALSE);
END_VAR

METHOD FB_init : BOOL
VAR_INPUT
	bInitRetains : BOOL; // if TRUE, the retain variables are initialized (warm start / cold start)
	bInCopyCode : BOOL;  // if TRUE, the instance afterwards gets moved into the copy code (online change)
END_VAR
AddParameter('in1', in1);
AddParameter('in2', in2);
AddOutput('out', out);
END_METHOD

METHOD PUBLIC  Clone : I_Node
VAR
	pNode : POINTER TO Node_XNOR;
END_VAR
pNode := __NEW(Node_XNOR);
Clone := pNode^;
END_METHOD

METHOD PROTECTED OnExecute
VAR
END_VAR
out.Value := NOT(in1.Value XOR in2.Value);
END_METHOD

END_FUNCTION_BLOCK

// Nodes/Logic/Node_XOR
{attribute 'linkalways'} 
{attribute 'no_explicit_call' := 'This FB is a CLASS and must be accessed using methods or properties'}
{attribute 'enable_dynamic_creation'}
FUNCTION_BLOCK FINAL Node_XOR EXTENDS Node
VAR
	in1 : _BOOL(FALSE);
    in2 : _BOOL(FALSE);
	out : _BOOL(FALSE);
END_VAR

METHOD FB_init : BOOL
VAR_INPUT
	bInitRetains : BOOL; // if TRUE, the retain variables are initialized (warm start / cold start)
	bInCopyCode : BOOL;  // if TRUE, the instance afterwards gets moved into the copy code (online change)
END_VAR
AddParameter('in1', in1);
AddParameter('in2', in2);
AddOutput('out', out);
END_METHOD

METHOD PUBLIC  Clone : I_Node
VAR
	pNode : POINTER TO Node_XOR;
END_VAR
pNode := __NEW(Node_XOR);
Clone := pNode^;
END_METHOD

METHOD PROTECTED OnExecute
VAR
END_VAR
out.Value := in1.Value XOR in2.Value;
END_METHOD

END_FUNCTION_BLOCK

// Nodes/TwinCAT/Node_TwinCATStatus
{attribute 'linkalways'} 
{attribute 'no_explicit_call' := 'This FB is a CLASS and must be accessed using methods or properties'}
{attribute 'enable_dynamic_creation'}
FUNCTION_BLOCK FINAL Node_TwinCATStatus EXTENDS Node
VAR
	lastCycleTime : _ULINT(0);
	averageCycleTime : _ULINT(0);
	usedMemory : _DWORD(0);
	avaliableMemory : _DWORD(0);
	maximumMemory : _DWORD(0);
	
	// node variables
	getRouterStatusInfo : FB_GetRouterStatusInfo;
	tcRouterStatusInfo : ST_TcRouterStatusInfo;
	cycleTimes : ARRAY [0..9] OF ULINT := [0,0,0,0,0,0,0,0,0,0];
    cycleTimeIndex : INT := 0;
END_VAR

METHOD FB_init : BOOL
VAR_INPUT
	bInitRetains : BOOL; // if TRUE, the retain variables are initialized (warm start / cold start)
	bInCopyCode : BOOL;  // if TRUE, the instance afterwards gets moved into the copy code (online change)
END_VAR
AddContent('lastCycleTime', lastCycleTime);
AddContent('averageCycleTime', averageCycleTime);
AddContent('usedMemory', usedMemory);
AddContent('avaliableMemory', avaliableMemory);
AddContent('maximumMemory', maximumMemory);
END_METHOD

METHOD PUBLIC  Clone : I_Node
VAR
	pNode : POINTER TO Node_TwinCATStatus;
END_VAR
pNode := __NEW(Node_TwinCATStatus);
Clone := pNode^;
END_METHOD

METHOD PROTECTED OnExecute
VAR
	i : INT;
    sum : ULINT := 0;
END_VAR
// memory 

IF NOT getRouterStatusInfo.bBusy THEN
	tcRouterStatusInfo := getRouterStatusInfo.info;
END_IF

getRouterStatusInfo(
	sNetId:= '' ,
	bExecute:= NOT getRouterStatusInfo.bBusy, 
	tTimeout:= T#5S, 
	bBusy=> , 
	bError=> , 
	nErrID=> , 
	info=> 
);

usedMemory.Value := tcRouterStatusInfo.maxMem - tcRouterStatusInfo.maxMemAvail;
avaliableMemory.Value := tcRouterStatusInfo.maxMemAvail;
maximumMemory.Value := tcRouterStatusInfo.maxMem;

// cycle time

cycleTimes[cycleTimeIndex] := F_GetTaskTotalTime(0);
cycleTimeIndex := (cycleTimeIndex + 1) MOD 10;

FOR i := 0 TO 9 DO
    sum := sum + cycleTimes[i];
END_FOR

lastCycleTime.Value := F_GetTaskTotalTime(0);
averageCycleTime.Value := sum / 10;
END_METHOD

END_FUNCTION_BLOCK

// Nodes/PlcNodePack
{attribute 'linkalways'} 
{attribute 'no_explicit_call' := 'This FB is a CLASS and must be accessed using methods or properties'}
{attribute 'enable_dynamic_creation'}
FUNCTION_BLOCK PlcNodePack
VAR
    // Conversion
	// DINT_TO
	node_DINT_TO_LREAL : Node_DINT_TO_LREAL;
	node_DINT_TO_REAL : Node_DINT_TO_REAL;
	// LREAL_TO_
	node_LREAL_TO_DINT : Node_LREAL_TO_DINT;
	node_LREAL_TO_UDINT : Node_LREAL_TO_UDINT;
	// REAL_TO_
    node_REAL_TO_DINT : Node_REAL_TO_DINT;
	node_REAL_TO_UDINT : Node_REAL_TO_UDINT;
	// UDINT_TO
	node_UDINT_TO_LREAL : Node_UDINT_TO_LREAL;
	node_UDINT_TO_REAL : Node_UDINT_TO_REAL;
    // Logic
    node_NOT : Node_NOT;
    node_AND : Node_AND;
    node_NAND : Node_NAND;
    node_OR : Node_OR;
    node_NOR : Node_NOR;
    node_XOR : Node_XOR;
    node_XNOR : Node_XNOR;
	
	// TwinCAT
	node_TwinCATStatus : Node_TwinCATStatus;
END_VAR

METHOD PUBLIC RegisterWithNodeFactory
VAR_INPUT
	NodeFactory : I_NodeFactory;
END_VAR
// Conversion
NodeFactory.AddNodeAsPrototype('PLC/Convert/DINT/DINT_TO_LREAL', node_DINT_TO_LREAL);
NodeFactory.AddNodeAsPrototype('PLC/Convert/DINT/DINT_TO_REAL', node_DINT_TO_REAL);
NodeFactory.AddNodeAsPrototype('PLC/Convert/LREAL/LREAL_TO_DINT', node_LREAL_TO_DINT);
NodeFactory.AddNodeAsPrototype('PLC/Convert/LREAL/LREAL_TO_UDINT', node_LREAL_TO_UDINT);
NodeFactory.AddNodeAsPrototype('PLC/Convert/REAL/REAL_TO_DINT', node_REAL_TO_DINT);
NodeFactory.AddNodeAsPrototype('PLC/Convert/REAL/REAL_TO_UDINT', node_REAL_TO_UDINT);
NodeFactory.AddNodeAsPrototype('PLC/Convert/UDINT/UDINT_TO_LREAL', node_UDINT_TO_LREAL);
NodeFactory.AddNodeAsPrototype('PLC/Convert/UDINT/UDINT_TO_REAL', node_UDINT_TO_REAL);

// Logic
NodeFactory.AddNodeAsPrototype('PLC/Logic/NOT', node_NOT);
NodeFactory.AddNodeAsPrototype('PLC/Logic/AND', node_AND);
NodeFactory.AddNodeAsPrototype('PLC/Logic/NAND', node_NAND);
NodeFactory.AddNodeAsPrototype('PLC/Logic/OR', node_OR);
NodeFactory.AddNodeAsPrototype('PLC/Logic/NOR', node_NOR);
NodeFactory.AddNodeAsPrototype('PLC/Logic/XOR', node_XOR);
NodeFactory.AddNodeAsPrototype('PLC/Logic/XNOR', node_XNOR);

// Hardware
//NodeFactory.AddNodeAsPrototype('PLC/Hardware/DI', node_DigitalInput);
//NodeFactory.AddNodeAsPrototype('PLC/Hardware/DO', node_DigitalOutput);

// TwinCAT
//NodeFactory.AddNodeAsPrototype('PLC/TwinCAT/TwinCAT Status', node_TwinCATStatus);
END_METHOD

END_FUNCTION_BLOCK

// PlcPack
{attribute 'linkalways'} 
{attribute 'no_explicit_call' := 'This FB is a CLASS and must be accessed using methods or properties'}
{attribute 'enable_dynamic_creation'}
FUNCTION_BLOCK PlcPack IMPLEMENTS I_GraphPack
VAR
	plcDatatypePack : PlcDatatypePack;
	plcNodePack : PlcNodePack;
END_VAR

METHOD Register
VAR_INPUT
	Datatypes : I_Datatypes;
	NodeFactory : I_NodeFactory;
END_VAR
plcDatatypePack.RegisterWithDatatypes(Datatypes);
plcNodePack.RegisterWithNodeFactory(NodeFactory);
END_METHOD

END_FUNCTION_BLOCK
